// TIA Portal V17 export
// export: Created 2024-06-14T09:53:55.4459219Z, ExportSetting WithDefaults, DisplayName Totally Integrated Automation Portal, DisplayVersion V17, DisplayName TIA Portal Openness, DisplayVersion V17, DisplayName TIA Portal Version Control Interface, DisplayVersion V17, DisplayName Simotion SCOUT TIA, DisplayVersion 5.4.3.0, DisplayName SINAMICS Startdrive Advanced, DisplayVersion V17 SP1 Update 1, DisplayName SINAMICS Startdrive G110M, G120, G120C, G120D, G120P, G115D, DisplayVersion V17 SP1 Update 1, DisplayName SINAMICS Startdrive G130, G150, S120, S150, SINAMICS MV, S210, DisplayVersion V17 SP1 Update 1, DisplayName STEP 7 Professional, DisplayVersion V17, DisplayName STEP 7 Safety, DisplayVersion V17, DisplayName WinCC Professional, DisplayVersion V17
TYPE "MODBUS_READ"
// stored: IsFailsafeCompliant false
   STRUCT
      MOD_COIL_DATA : Array[1..32] of Bool;
      MOD_HOLD_DATA_1 : Array[1..6] of Word;
      MOD_HOLD_DATA_2 : Array[1..2] of Word;
   END_STRUCT;
   // // MOD_COIL_DATA[1] : Satble Flag
   // // MOD_COIL_DATA[2] : Net Gross Flag
   // // MOD_COIL_DATA[3] : Operating Mode
   // // MOD_COIL_DATA[4] : Start Key Status
   // // MOD_COIL_DATA[5] : Zero Key Status
   // // MOD_COIL_DATA[6] : Tare Key Status
   // // MOD_COIL_DATA[7] : Print Key Status
   // // MOD_COIL_DATA[8] : Power On Zero
   // // MOD_COIL_DATA[9] : One Touch Zero Calibration
   // // MOD_COIL_DATA[10] : Under Weight Flag
   // // MOD_COIL_DATA[11] : Over Weight Flag
   // // MOD_COIL_DATA[12] : Gross Sign
   // // MOD_COIL_DATA[13] : Net Sign
   // // MOD_COIL_DATA[14] : Filled or Checked Data Status(W)
   // // MOD_COIL_DATA[15] : NA
   // // MOD_COIL_DATA[16] : Gate Input
   // // MOD_COIL_DATA[17] : Coarse Output
   // // MOD_COIL_DATA[18] : Fine Output
   // // MOD_COIL_DATA[19] : Batch Over Output
   // // MOD_COIL_DATA[20] : Gate Output
   // // MOD_COIL_DATA[21] : Lifter Output
   // // MOD_COIL_DATA[22] : Jam Output
   // // MOD_COIL_DATA[23] : NA
   // // MOD_COIL_DATA[24] : Indicator is in Parameter / Tare Entry Settings
   // // MOD_COIL_DATA[25] : Filling ON Status
   // // MOD_COIL_DATA[26] : Filling Time Over (W)
   // // MOD_COIL_DATA[27] : Tare Request Status
   // // MOD_COIL_DATA[28] : Filling Over Status
   // // MOD_COIL_DATA[29] : Filling Error Status(W)
   // // MOD_COIL_DATA[30] : Stop Filling (W)
   // // MOD_COIL_DATA[31] : Start Filling (W)
   // // MOD_COIL_DATA[32] : Tare Entry Error
   // // MOD_HOLD_DATA_1[2] : Fiiled Gross Weight
   // // MOD_HOLD_DATA_1[4] : Filled Net Weight
   // // MOD_HOLD_DATA_1[6] : Punched Tare Weight
   // // MOD_HOLD_DATA_2[2] : Fiiled Gross Weight
END_TYPE
